PROGRAM Permissives
VAR
	i : INT := 1;  //for section 1 - 3 
	j : INT := 1; //for charger 1-8
	
END_VAR

//Charger summary faults
//Trips_DB.AnySummaryFault = FALSE AND Trips_DB.AnyEstopPressed //add to no fault detected.

//section ready to charge
FOR i := 1 TO 3 BY 1 DO
	IF Trips_DB.NoFaultDetected = TRUE AND //MCP_IO.Charger[1-8].HVisOn AND
		Permissives_DB.AllChargeRelaysClosed = TRUE AND
		LCP.Section[i].Peak.ShortContactEngaged = FALSE AND
		LCP.Section[i].Sust.ShortContactEngaged = FALSE
	THEN
		LCP.Section[i].SystemReadyToCharge := TRUE;	
	ELSE
		LCP.Section[i].SystemReadyToCharge := FALSE;		
	END_IF;
END_FOR;

//Section 4
IF Trips_DB.NoFaultDetected = TRUE AND //MCP_IO.Charger[1-8].HVisOn AND
	Permissives_DB.AllChargeRelaysClosed = TRUE AND
	LCP.Section[4].Form.ShortContactEngaged = FALSE AND
	LCP.Section[4].Form.FormTrigShortContactEngaged = FALSE AND
	LCP.Section[4].Form.PreFormTrigShortContactEngaged = FALSE 
	THEN
		LCP.Section[4].SystemReadyToCharge := TRUE;
	ELSE
		LCP.Section[4].SystemReadyToCharge := FALSE;
END_IF;
	



// shorts and unshorts
//Peaking  -- short contacts are NO, so if close is false, it is and unshort is true, then it is not shorted 
FOR i := 1 TO 3 BY 1 DO
	IF LCP.Section[i].Peak.ShortContact1_close = FALSE AND LCP.Section[i].Peak.UnshortContact1_close = TRUE AND
		LCP.Section[i].Peak.ShortContact2_close = FALSE AND LCP.Section[i].Peak.UnshortContact2_close = TRUE 
		THEN
			LCP.Section[i].Peak.ShortContactEngaged := FALSE;
		ELSE
			LCP.Section[i].Peak.ShortContactEngaged := TRUE;
	END_IF;
END_FOR;

//Sustain
FOR i := 1 TO 3 BY 1 DO
	IF LCP.Section[i].Sust.ShortContact1_close = FALSE AND LCP.Section[i].Sust.UnshortContact1_close = TRUE AND
		LCP.Section[i].Sust.ShortContact2_close = FALSE AND LCP.Section[i].Sust.UnshortContact2_close = TRUE 
		THEN
			LCP.Section[i].Sust.ShortContactEngaged := FALSE;
		ELSE
			LCP.Section[i].Sust.ShortContactEngaged := TRUE;
	END_IF;
END_FOR;

//Formation
IF LCP.Section[4].Form.ShortContact1_close = FALSE AND LCP.Section[4].Form.UnshortContact1_close = TRUE AND
	LCP.Section[4].Form.ShortContact2_close = FALSE AND LCP.Section[4].Form.UnshortContact2_close = TRUE 
	THEN
		LCP.Section[4].Form.ShortContactEngaged := FALSE;
	ELSE
		LCP.Section[4].Form.ShortContactEngaged := TRUE; //might need to clarify on the NC of the short contacts.
END_IF;
// form trig short 
IF LCP.Section[4].Form.FormTrigShortContact_close = FALSE AND LCP.Section[4].Form.FormTrigUnShortContact_close = TRUE
	THEN
		LCP.Section[4].Form.FormTrigShortContactEngaged := FALSE;
	ELSE
		LCP.Section[4].Form.FormTrigShortContactEngaged := TRUE;
END_IF
// preform trig short 
IF LCP.Section[4].Form.PreFormTrigShortContact_close = FALSE AND LCP.Section[4].Form.PreFormTrigUnShortContact_close = TRUE
	THEN
		LCP.Section[4].Form.PreFormTrigShortContactEngaged := FALSE;
	ELSE
		LCP.Section[4].Form.PreFormTrigShortContactEngaged := TRUE;
END_IF

//any short contact engaged

IF LCP.Section[1].Peak.ShortContactEngaged = TRUE AND 
	LCP.Section[2].Peak.ShortContactEngaged = TRUE AND
	LCP.Section[3].Peak.ShortContactEngaged = TRUE AND
	LCP.Section[1].Sust.ShortContactEngaged = TRUE AND
	LCP.Section[2].Sust.ShortContactEngaged = TRUE AND 
	LCP.Section[3].Sust.ShortContactEngaged = TRUE AND 
	LCP.Section[4].Form.ShortContactEngaged = TRUE AND 
	LCP.Section[4].Form.FormTrigShortContactEngaged = TRUE AND //
	LCP.Section[4].Form.PreFormTrigShortContactEngaged = TRUE //
	THEN
		Permissives_DB.AllShortContactEngaged := TRUE;
	ELSE 
		Permissives_DB.AllShortContactEngaged := FALSE;	
END_IF;

//All charger inhibited
IF MCP_IO.Charger[1].inhibited = TRUE AND
	MCP_IO.Charger[2].inhibited = TRUE AND
	MCP_IO.Charger[3].inhibited = TRUE AND
	MCP_IO.Charger[4].inhibited = TRUE AND
	MCP_IO.Charger[5].inhibited = TRUE AND
	MCP_IO.Charger[6].inhibited = TRUE AND
	MCP_IO.Charger[7].inhibited = TRUE AND
	MCP_IO.Charger[8].inhibited = TRUE 
	THEN
		MCP_IO.AllChargerInhibited := TRUE;
		ELSE
			MCP_IO.AllChargerInhibited := FALSE;
END_IF;

//All charger HV ON
IF MCP_IO.Charger[1].HV_isON = TRUE AND
	MCP_IO.Charger[2].HV_isON = TRUE AND
	MCP_IO.Charger[3].HV_isON = TRUE AND
	MCP_IO.Charger[4].HV_isON = TRUE AND
	MCP_IO.Charger[5].HV_isON = TRUE AND
	MCP_IO.Charger[6].HV_isON = TRUE AND
	MCP_IO.Charger[7].HV_isON = TRUE AND
	MCP_IO.Charger[8].HV_isON = TRUE 
	THEN
		MCP_IO.AllChargerHVisON := TRUE;
		ELSE
			MCP_IO.AllChargerHVisON := FALSE;
END_IF;


//All charge relay close
IF LCP.Section[1].Peak.ChargeRelay1_close = TRUE AND
	LCP.Section[1].Peak.ChargeRelay2_close = TRUE AND
	LCP.Section[1].Sust.ChargeRelay1_close = TRUE AND
	LCP.Section[1].Sust.ChargeRelay2_close = TRUE AND
	LCP.Section[2].Peak.ChargeRelay1_close = TRUE AND
	LCP.Section[2].Peak.ChargeRelay2_close = TRUE AND
	LCP.Section[2].Sust.ChargeRelay1_close = TRUE AND
	LCP.Section[2].Sust.ChargeRelay2_close = TRUE AND
	LCP.Section[3].Peak.ChargeRelay1_close = TRUE AND
	LCP.Section[3].Peak.ChargeRelay2_close = TRUE AND
	LCP.Section[3].Sust.ChargeRelay1_close = TRUE AND
	LCP.Section[3].Sust.ChargeRelay2_close = TRUE AND
	
	LCP.Section[4].Form.ChargeRelay1_close = TRUE AND
	LCP.Section[4].Form.ChargeRelay2_close = TRUE AND						
	LCP.Section[4].Form.PreFormChargeRly_close = TRUE AND
	LCP.Section[4].Form.FormTrigChargeRly_close = TRUE AND
	LCP.Section[4].Form.PreFormTrigChargeRly_close = TRUE 
	THEN
		Permissives_DB.AllChargeRelaysClosed := TRUE;
	ELSE
		Permissives_DB.AllChargeRelaysClosed := FALSE;
END_IF;

//All Dump relays open  ******
IF LCP.Section[1].Peak.DumpRelay1_close = FALSE AND
	LCP.Section[1].Peak.DumpRelay2_close = FALSE AND
	LCP.Section[1].Sust.DumpRelay1_close = FALSE AND
	LCP.Section[1].Sust.DumpRelay2_close = FALSE AND
	LCP.Section[2].Peak.DumpRelay1_close = FALSE AND
	LCP.Section[2].Peak.DumpRelay2_close = FALSE AND
	LCP.Section[2].Sust.DumpRelay1_close = FALSE AND
	LCP.Section[2].Sust.DumpRelay2_close = FALSE AND
	LCP.Section[3].Peak.DumpRelay1_close = FALSE AND
	LCP.Section[3].Peak.DumpRelay2_close = FALSE AND
	LCP.Section[3].Sust.DumpRelay1_close = FALSE AND
	LCP.Section[3].Sust.DumpRelay2_close = FALSE AND
	
	LCP.Section[4].Form.DumpRelay1_close = FALSE AND
	LCP.Section[4].Form.DumpRelay2_close = FALSE AND						
	LCP.Section[4].Form.PreFormDumpRly_close = FALSE AND
	LCP.Section[4].Form.FormTrigDumpRly1_close = FALSE AND
	LCP.Section[4].Form.PreFormTrigDumpRly1_close = FALSE 
	THEN
		Permissives_DB.AllDumpRelaysOpen := TRUE;
	ELSE
		Permissives_DB.AllDumpRelaysOpen := FALSE;
END_IF;


IF i > 3 THEN
	i := 1;
END_IF;


IF j > 8 THEN
	j := 1;
END_IF;

END_PROGRAM

(* stored: Version 1.1.0.1, ProductVersion 3.1.4024.11
   POU Permissives: Id {a037c57d-7935-4b17-bb0a-42e72a6c09c9}, SpecialFunc None *)
